// Block: F_DB

DATA_BLOCK F_DB
VERSION : 0.1
   NON_RETAIN
   VAR
      SafetyReset : Bool;
      SuperUserReset : Bool;
      Enable_Reset_Superuser : Bool;
      A01_Estop : Bool;
      A01_EstopDelay : Bool;
      A02_Estop : Bool;
      A02_EstopDelay : Bool;
      A03_Estop : Bool;
      A03_EstopDelay : Bool;
      LB101 : udt_BimanualSts;
      LB111 : udt_BimanualSts;
      LB112 : udt_BimanualSts;
      LB113 : udt_BimanualSts;
      LB113_W : udt_BimanualSts;
      LB114_FeedA01 : udt_BimanualSts;
      LB114_FeedA02 : udt_BimanualSts;
      LB131 : udt_BimanualSts;
      LB211 : udt_BimanualSts;
      LB212 : udt_BimanualSts;
      LB212_FeedA02 : udt_BimanualSts;
      LB311 : udt_BimanualSts;
      D01 : udt_DoorSts;
      D02 : udt_DoorSts;
      D03 : udt_DoorSts;
      D04 : udt_DoorSts;
      D05 : udt_DoorSts;
      D07 : udt_DoorSts;
      D10 : udt_DoorSts;
      D11 : udt_DoorSts;
      D12 : udt_DoorSts;
      D14 : udt_DoorSts;
      D15 : udt_DoorSts;
      D16 : udt_DoorSts;
      D18 : udt_DoorSts;
      D19 : udt_DoorSts;
      D20 : udt_DoorSts;
      D21 : udt_DoorSts;
      D22 : udt_DoorSts;
      D24 : udt_DoorSts;
      D25 : udt_DoorSts;
      D27 : udt_DoorSts;
      D30 : udt_DoorSts;
      ZSI_Zone00 : udt_ZoneSafetyInterface;
      ZSI_Zone01 : udt_ZoneSafetyInterface;
      ZSI_Zone02 : udt_ZoneSafetyInterface;
      ZSI_Zone03 : udt_ZoneSafetyInterface;
      ZSI_Zone05 : udt_ZoneSafetyInterface;
      ZSI_Zone06 : udt_ZoneSafetyInterface;
      ZSI_Zone10 : udt_ZoneSafetyInterface;
      ZSI_Zone11 : udt_ZoneSafetyInterface;
      ZSI_Zone13 : udt_ZoneSafetyInterface;
      ZSI_Zone15 : udt_ZoneSafetyInterface;
      ZSI_Zone20 : udt_ZoneSafetyInterface;
      ZSI_Zone21 : udt_ZoneSafetyInterface;
      ZSI_Zone23 : udt_ZoneSafetyInterface;
      ZSI_Zone25 : udt_ZoneSafetyInterface;
      ZSI_Zone27 : udt_ZoneSafetyInterface;
      ZSI_Zone29 : udt_ZoneSafetyInterface;
      FNS_Zone05 : Bool;
      FNS_Zone10 : Bool;
      FNS_Zone11 : Bool;
      FNS_Zone13 : Bool;
      FNS_Zone15 : Bool;
      FNS_Zone20 : Bool;
      FNS_Zone21 : Bool;
      FNS_Zone23 : Bool;
      FNS_Zone25 : Bool;
      FNS_Zone27 : Bool;
      FNS_Zone29 : Bool;
      DSI_V_Air_Gen : udt_DeviceSafetyInterface;
      DSI_S120_CoilCar : udt_DeviceSafetyInterface;
      DSI_V_CoilCar : udt_DeviceSafetyInterface;
      DSI_HU_Decoilers_Pump : udt_DeviceSafetyInterface;
      DSI_S120_Decoiler1 : udt_DeviceSafetyInterface;
      DSI_V_Decoiler1 : udt_DeviceSafetyInterface;
      DSI_S120_Decoiler2 : udt_DeviceSafetyInterface;
      DSI_V_Decoiler2 : udt_DeviceSafetyInterface;
      DSI_S120_DecoilersTranslation : udt_DeviceSafetyInterface;
      DSI_V_DecoilersHorizRotation : udt_DeviceSafetyInterface;
      DSI_HU_Area01_Pump : udt_DeviceSafetyInterface;
      DSI_V_Peeler : udt_DeviceSafetyInterface;
      DSI_S120_Straightener : udt_DeviceSafetyInterface;
      DSI_V_JB_Cut_Rest : udt_DeviceSafetyInterface;
      DSI_V_JB_Cut_Work : udt_DeviceSafetyInterface;
      DSI_S120_JB_Torch : udt_DeviceSafetyInterface;
      DSI_S120_JB_PinchRoll : udt_DeviceSafetyInterface;
      DSI_S120_Rollformer : udt_DeviceSafetyInterface;
      DSI_S120_Cassetta1_OP : udt_DeviceSafetyInterface;
      DSI_S120_Cassetta1_MOT : udt_DeviceSafetyInterface;
      DSI_S120_Cassetta2_OP : udt_DeviceSafetyInterface;
      DSI_S120_Cassetta2_MOT : udt_DeviceSafetyInterface;
      DSI_S120_Cassetta3_OP : udt_DeviceSafetyInterface;
      DSI_S120_Cassetta3_MOT : udt_DeviceSafetyInterface;
      DSI_S120_FAK_Pusher : udt_DeviceSafetyInterface;
      DSI_S120_Carriage : udt_DeviceSafetyInterface;
      DSI_S120_AccRolls1 : udt_DeviceSafetyInterface;
      DSI_S120_AccRolls2 : udt_DeviceSafetyInterface;
      DSI_S120_AccRolls3 : udt_DeviceSafetyInterface;
      DSI_HU_FinalCut_Pump : udt_DeviceSafetyInterface;
      DSI_V_FinalCut : udt_DeviceSafetyInterface;
      DSI_CambioFormato_Profilatrice : udt_DeviceSafetyInterface;
      DSI_V_Air_A0301_A0302 : udt_DeviceSafetyInterface;
      DSI_Trasporto : udt_DeviceSafetyInterface;
      DSI_Ribaltatore : udt_DeviceSafetyInterface;
      DSI_Spintore : udt_DeviceSafetyInterface;
      DSI_S120_Bordatrice : udt_DeviceSafetyInterface;
      DSI_CambioFormato_Bordatrice : udt_DeviceSafetyInterface;
      DSI_V_Air_A0302_A0303 : udt_DeviceSafetyInterface;
      DSI_Rulliera1 : udt_DeviceSafetyInterface;
      DSI_Rulliera2 : udt_DeviceSafetyInterface;
      DSI_HU_CYTROPAC_STO : udt_DeviceSafetyInterface;
      DSI_V_PareggiatoreCoda : udt_DeviceSafetyInterface;
      DSI_V_PareggiatoreTesta : udt_DeviceSafetyInterface;
      DSI_PareggiatoreTesta : udt_DeviceSafetyInterface;
      DSI_PareggiatoreCoda : udt_DeviceSafetyInterface;
      DSI_ManipolatoreTesta : udt_DeviceSafetyInterface;
      DSI_ManipolatoreCoda : udt_DeviceSafetyInterface;
      DSI_SpallaTesta : udt_DeviceSafetyInterface;
      DSI_SpallaCoda : udt_DeviceSafetyInterface;
      DSI_TraslazioneTesta : udt_DeviceSafetyInterface;
      DSI_TraslazioneCoda : udt_DeviceSafetyInterface;
      DSI_SollevamentoTesta : udt_DeviceSafetyInterface;
      DSI_SollevamentoCoda : udt_DeviceSafetyInterface;
      DSI_SostegnoAntiribCoda : udt_DeviceSafetyInterface;
      DSI_SostegnoAntiribTesta : udt_DeviceSafetyInterface;
      DSI_V_Air_A0304 : udt_DeviceSafetyInterface;
      DSI_NavettaTesta : udt_DeviceSafetyInterface;
      DSI_NavettaCoda : udt_DeviceSafetyInterface;
   END_VAR

BEGIN
   // No initialization required
END_DATA_BLOCK
